# EPICS substitutions: apps/jscalerApp/Db/jscalers_TDCFTOF2_TRIG.substitutions
file "db/jscaler_channel.db" {
pattern { CrNo,CrName,Sl,Ch,Det,Sys,Element,CScode,Thresh,Mode,Counts }
{ "05","TDCFTOF2","20","15","TRIG","CAEN","SEC2_A","5125","15","271","15" }
}
